FUNCTION_BLOCK FB_Warmtepomp
VAR
	Verbruik		: FB_Verbruikmeter;
	Communicatie	: Warmtepomp_Signalen;
	
END_VAR

END_FUNCTION_BLOCK

(* stored: Version 1.1.0.1, ProductVersion 3.1.4024.12
   POU FB_Warmtepomp: Id {a009efd3-353e-4f00-aa50-3faa99f6125b}, SpecialFunc None *)
